INTERFACE IStringBuilder

METHOD  Append : IStringBuilder // Append text to t current build string.
VAR_INPUT
	text:STRING; //Text to append to current build string
END_VAR
END_METHOD

METHOD InsertAtLocation : IStringBuilder
VAR_INPUT
	Text:STRING;
	Position:INT;
END_VAR
END_METHOD

METHOD Reset : ILimitedStringBuilder //Reset current build string to an empty string.
END_METHOD

METHOD ToString : STRING //Returns current build string.
END_METHOD

END_INTERFACE

(* stored: Version 1.1.0.1, ProductVersion 3.1.4024.0
   Itf IStringBuilder: Id {cc6d396c-ab11-4512-b217-fcaa420ac27e}
   Method Append: Id {39f6182f-ddaa-4a04-88e3-b41671a4f64d}
   Method InsertAtLocation: Id {84b072e0-2852-4c7d-a45f-8bbe495344a7}
   Method Reset: Id {6ef3d071-ad38-492e-ac0f-193eb38816d5}
   Method ToString: Id {857ec4df-c977-46b4-ad47-ee4fdd52fb44} *)
